// note: 17 stored wires end on pins the file does not list and are not shown
IF NOT (HW_ACV.Mode=Burkert.eACV_Modes.Auto) THEN _w1 := Mix_Status.HW_Valve_Not_Ready; END_IF
Control.Status := _w1;
IF NOT (CW_ACV.Mode=Burkert.eACV_Modes.Auto) THEN _w2 := Mix_Status.CW_Valve_Not_Ready; END_IF
Control.Status := _w2;
Control.Actual_Rate_EU := FIT.Rate;
_w3 := (Control.Mode=Mix_Modes.IDlE) OR (Control.STATUS>Mix_Status.Batch_Ending) OR (Control.Mode=Mix_Modes.Pause);
RATE_PID(
    ACT := FIT.Rate,
    SET := Live_Rate,
    SUP := 0.1,
    OFS := 0.0,
    M_I := 0.0,
    MAN := _w3,
    RST := _w3,
    KP := Control.Config.Flow_KP,
    TN := Control.Config.Flow_TN,
    TV := Control.Config.Flow_TV,
    LL := 0,
    LH := 100.0); // BURKERT_OSCAT_BASIC.CTRL_PID
Control.Flow_CV := RATE_PID.Y;
R_TRIG_2(CLK := _w3 AND (Temperature.Mode.eMode<>Burkert.AIT_Modes.Forced)); // R_Trig
IF R_TRIG_2.Q THEN _w4 := Burkert.AIT_Modes.Alarms_Disabled; END_IF
Temperature.Mode.eMode := _w4;
Control.Actual_Temp_EU := Temperature.EU;
_w5 := (Control.Mode=Mix_Modes.IDlE) OR (Control.Mode=Mix_Modes.Rate_Only) OR (Control.STATUS>Mix_Status.Batch_Ending) OR (Control.STATUS=Mix_Status.Start_Flow) OR (Control.STATUS=Mix_Status.Fit_Reset) OR (Control.Mode=Mix_Modes.Pause);
PID_0(
    ACTUAL := Temperature.EU,
    SET_POINT := Control.Config.TARGET_C,
    KP := Control.Config.Temp_KP,
    TN := Control.Config.Temp_TN,
    TV := Control.Config.Temp_TV,
    Y_MANUAL := 0,
    Y_OFFSET := 0,
    Y_MIN := -100,
    Y_MAX := 100,
    MANUAL := _w5,
    RESET := _w5); // Util.PID
Control.Temp_CV := SEl(Control.Mode=Mix_Modes.Cold_Only, SEl(Control.Mode=Mix_Modes.Hot_Only, PID_0.Y, 100), -100);
SRAMP_0(
    X := Ramp_Target,
    A_UP := Control.Config.Ramp_Rate,
    A_DN := 0-Control.config.Ramp_Rate,
    VU_MAX := Control.config.Max_Flow,
    VD_MAX := 0-Control.config.Max_Flow,
    LIMIT_HIGH := Control.config.Max_Flow,
    LIMIT_LOW := Control.Config.Min_Flow,
    RST := Control.Mode=Mix_Modes.IDlE); // BURKERT_OSCAT_BASIC.SRAMP
Live_Rate := SRAMP_0.Y;
IF Control.Mode=Mix_Modes.IDlE THEN _w6 := Mix_Status.IDle; END_IF
Control.STATUS := _w6;
R_TRIG_0(CLK := (Control.Mode=Mix_Modes.Auto) OR (Control.Mode=Mix_Modes.Hot_Only) OR (Control.Mode=Mix_Modes.Cold_Only) OR (Control.Mode=Mix_Modes.Quick_Start)); // R_Trig
Control.STATUS := SEL(R_TRIG_0.Q, Control.STATUS, Mix_Status.Fit_Reset);
Control.Actual_Volume_EU := FIT.Total;
_w7 := Control.STATUS = Mix_Status.Fit_Reset;
IF _w7 THEN _w8 := False; END_IF
Ramp_active := _w8;
_w9 := NOT (FIT.Total>0.1) AND _w7;
FIT.PLC_Reset := SEL(_w7 AND (FIT.Total>0.1), SEL(_w9, FIT.PLC_Reset, False), True);
_w10 := _w9;
IF _w10 THEN _w11 := Mix_Status.Start_Flow; END_IF
_w12 := _w10;
IF _w12 THEN _w13 := SEL(Control.Mode=Mix_Modes.Hot_Only, _w11, Mix_Status.Temperature_OK); END_IF
IF _w12 THEN _w14 := SEL(Control.Mode=Mix_Modes.Hot_Only, _w13, Mix_Status.Temperature_OK); END_IF
Control.STATUS := _w14;
_w15 := Control.Temp_CV / 100.0;
_w16 := LIMIT(0, Control.Flow_CV * (1.0 + _w15), 100);
Control.HW_CMD := _w16;
HW_ACV.PLC_CMD := _w16;
_w17 := LIMIT(0, Control.Flow_CV * (1.0 - _w15), 100);
Control.CW_CMD := _w17;
CW_ACV.PLC_CMD := _w17;
_w18 := Control.STATUS = Mix_Status.Start_Flow;
IF _w18 THEN _w19 := Control.Config.Min_Flow; END_IF
Ramp_Target := _w19;
TON_0(IN := _w18 AND (Control.Actual_Rate_EU > (Control.Config.Min_Flow*0.8) OR (Control.Mode=Mix_Modes.Quick_Start)), PT := Stage_Delay); // TON
Control.STATUS := SEL(TON_0.Q, Control.STATUS, Mix_Status.Flow_Detected);
TON_1(IN := Control.STATUS = Mix_Status.Flow_Detected, PT := Stage_Delay); // TON
R_TRIG_3(CLK := (Temperature.Mode.eMode<>Burkert.AIT_Modes.Forced) AND TON_1.Q); // R_Trig
IF R_TRIG_3.Q THEN _w20 := Burkert.TT_Modes.Active; END_IF
Temperature.Mode.eMode := _w20;
Control.STATUS := SEL(TON_1.Q, Control.STATUS, Mix_Status.Start_temperature);
Temperature.Burkert.cAlarm_Config.Hi_Hi_Alarm := Control.Config.TARGET_C+(Control.Config.TEMP_WINDOW*4);
Temperature.Burkert.cAlarm_Config.Hi_Warn := Control.Config.TARGET_C+(Control.Config.TEMP_WINDOW*2);
Temperature.Burkert.cAlarm_Config.Low_warn := Control.Config.TARGET_C-(Control.Config.TEMP_WINDOW*2);
Temperature.Burkert.cAlarm_Config.Low_Low_Alarm := Control.Config.TARGET_C-(Control.Config.TEMP_WINDOW*4);
TON_2(IN := Control.STATUS = Mix_Status.Start_temperature AND (Control.Actual_Temp_EU > (Control.Config.TARGET_C-Control.Config.TEMP_WINDOW) OR (Control.Mode=Mix_Modes.Quick_Start)), PT := Stage_Delay); // TON
Control.STATUS := SEL(TON_2.Q, Control.STATUS, Mix_Status.Temperature_OK);
TON_3(IN := Control.STATUS = Mix_Status.Temperature_OK, PT := Stage_Delay); // TON
Control.STATUS := SEL(TON_3.Q, Control.STATUS, Mix_Status.Foundation_Rate);
_w21 := Control.STATUS = Mix_Status.Foundation_Rate;
Ramp_Active := SEL(_w21, Ramp_Active, True);
_w22 := _w21;
IF _w22 THEN _w23 := Control.Config.Foundation_Rate; END_IF
Ramp_Target := _w23;
Control.STATUS := SEL(_w22 AND (Control.Actual_Rate_EU >= (Control.Config.Foundation_Rate*0.9) OR (Control.Mode=Mix_Modes.Quick_Start)), Control.STATUS, Mix_Status.Foundation_Rate_OK);
TON_4(IN := Control.STATUS = Mix_Status.Foundation_Rate_OK AND (FIT.Total >= Control.Config.Foundation_Volume OR (Control.Mode=Mix_Modes.Quick_Start)), PT := Stage_Delay); // TON
Control.STATUS := SEL(TON_4.Q, Control.STATUS, Mix_Status.Foundation_Amount_Complete);
R_TRIG_5(CLK := Control.Mode=Mix_Modes.Resume); // R_trig
TON_5(IN := Control.STATUS = Mix_Status.Foundation_Amount_Complete, PT := Stage_Delay); // TON
Control.STATUS := SEL(R_TRIG_5.Q OR TON_5.Q, Control.STATUS, Mix_Status.Main_Rate);
_w24 := Control.STATUS = Mix_Status.Main_Rate;
R_TRIG_1(CLK := _w24); // R_trig
IF R_TRIG_1.Q THEN _w25 := Control.Actual_Volume_EU; END_IF
Ramp_Start_Volume := _w25;
_w26 := _w24;
IF _w26 THEN _w27 := Control.Config.TARGET_lpm; END_IF
Ramp_Target := _w27;
_w28 := _w26 AND Control.Actual_Rate_EU >= (Control.Config.TARGET_lpm*0.9);
Control.STATUS := SEL(_w28, Control.STATUS, Mix_Status.Main_Rate_OK);
IF _w28 THEN _w29 := Control.Actual_Volume_EU - Ramp_Start_Volume; END_IF
Ramp_Volume := _w29;
_w30 := Control.STATUS = Mix_Status.Main_Rate_OK;
TON_6(IN := _w30, PT := Stage_Delay); // TON
Control.STATUS := SEL(TON_6.Q, Control.STATUS, Mix_Status.Grain_Dispense);
_w31 := Control.STATUS = Mix_Status.Grain_Dispense;
_w32 := _w31;
IF _w32 THEN _w33 := Control.Config.TARGET_C; END_IF
Control.Config.TARGET_C := _w33;
IF _w32 THEN _w34 := Control.Config.TARGET_lpm; END_IF
Ramp_Target := _w34;
Control.STATUS := SEL(_w31 AND Control.Actual_Volume_EU >= (Control.Config.TARGET_L-Control.Config.Foundation_Volume), Control.STATUS, Mix_Status.Batch_Ending);
IF Control.Actual_Rate_EU>0.5 THEN _w35 := ((Control.Config.TARGET_L-Control.Config.Foundation_Volume) - Control.Actual_Volume_EU) / (Control.Actual_Rate_EU/60); END_IF
Control.Grain_ETA_S := REAL_TO_INT(_w35);
_w36 := Control.STATUS = Mix_Status.Batch_Ending;
IF _w36 THEN _w37 := Control.Config.Foundation_Rate; END_IF
Ramp_Target := _w37;
_w38 := (_w24 OR _w30 OR _w31 OR _w36) AND Control.Actual_Volume_EU >= Control.Config.TARGET_L;
Ramp_Active := SEl(_w38, Ramp_Active, FALSE);
Control.STATUS := SEL(_w38, Control.STATUS, Mix_Status.Batch_Complete);
// 0.1: input not connected

END_FUNCTION_BLOCK

// Tempered_Mix_UDFB
FUNCTION_BLOCK Tempered_Mix_UDFB
VAR_INPUT
	//Loop_ID:INT;
END_VAR
VAR_IN_OUT
	HW_ACV:Burkert.cACV;
	CW_ACV:Burkert.cACV;
	Temperature:Burkert.cSensor;
	FIT:Burkert.cFIT;
	Control:Mix_DUT;
END_VAR
VAR_OUTPUT
END_VAR
VAR
	R_TRIG_0: R_Trig;
	RATE_PID: BURKERT_OSCAT_BASIC.CTRL_PID;
	
	Temp_PID: BURKERT_OSCAT_BASIC.CTRL_PID;
	TON_0: TON;
	Stage_Delay: TIME := T#2s;
	TON_1: TON;
	TON_2: TON;
	SRAMP_0: BURKERT_OSCAT_BASIC.SRAMP;
	TON_3: TON;
	TON_4: TON;
	Ramp_Active: BOOL;
	Ramp_Target: REAL;
	TON_5: TON;
	TON_6: TON;
	R_TRIG_1: R_trig;
	Ramp_Start_Volume: REAL;
	Ramp_Volume: REAL;
	R_TRIG_2: R_Trig;
	R_TRIG_3: R_Trig;
	PID_0: Util.PID;
	R_TRIG_4: R_Trig;
	R_TRIG_5:R_trig;
	
	Live_Rate: REAL;
END_VAR
VAR // added by the converter: edge detectors and wires of the graphical bodies
    _w1, _w2, _w3, _w4, _w5, _w6, _w10, _w12, _w13, _w14, _w15, _w16, _w18, _w19, _w21, _w23, _w25, _w30, _w32 : ANY;
    _w7, _w8, _w9, _w11, _w17, _w20, _w22, _w24, _w26, _w28, _w29, _w31, _w33 : BOOL;
    _w27 : REAL;
END_VAR

// note: 18 stored wires end on pins the file does not list and are not shown
IF NOT (HW_ACV.Mode.eMode=Burkert.eACV_Modes.Auto) THEN _w1 := Mix_Status.HW_Valve_Not_Ready; END_IF
Control.Status := _w1;
IF NOT (CW_ACV.Mode.eMode=Burkert.eACV_Modes.Auto) THEN _w2 := Mix_Status.CW_Valve_Not_Ready; END_IF
Control.Status := _w2;
Control.Actual_Rate_EU := FIT.Rate.EU;
_w3 := (Control.Mode=Mix_Modes.IDlE) OR (Control.STATUS>Mix_Status.Batch_Ending) OR (Control.Mode=Mix_Modes.Pause);
RATE_PID(
    ACT := FIT.Rate.EU,
    SET := Live_Rate,
    SUP := 0.1,
    OFS := 0.0,
    M_I := 0.0,
    MAN := _w3,
    RST := _w3,
    KP := Control.Config.Flow_KP,
    TN := Control.Config.Flow_TN,
    TV := Control.Config.Flow_TV,
    LL := 0,
    LH := 100.0); // BURKERT_OSCAT_BASIC.CTRL_PID
Control.Flow_CV := RATE_PID.Y;
R_TRIG_2(CLK := _w3 AND (Temperature.Mode.eMode<>Burkert.AIT_Modes.Forced)); // R_Trig
IF R_TRIG_2.Q THEN _w4 := Burkert.AIT_Modes.Alarms_Disabled; END_IF
Temperature.Mode.eMode := _w4;
Control.Actual_Temp_EU := Temperature.EU;
_w5 := (Control.Mode=Mix_Modes.IDlE) OR (Control.Mode=Mix_Modes.Rate_Only) OR (Control.STATUS>Mix_Status.Batch_Ending) OR (Control.STATUS=Mix_Status.Start_Flow) OR (Control.STATUS=Mix_Status.Fit_Reset) OR (Control.Mode=Mix_Modes.Pause);
PID_0(
    ACTUAL := Temperature.EU,
    SET_POINT := Control.Config.TARGET_C,
    KP := Control.Config.Temp_KP,
    TN := Control.Config.Temp_TN,
    TV := Control.Config.Temp_TV,
    Y_MANUAL := 0,
    Y_OFFSET := 0,
    Y_MIN := -100,
    Y_MAX := 100,
    MANUAL := _w5,
    RESET := _w5); // Util.PID
Control.Temp_CV := SEl(Control.Mode=Mix_Modes.Cold_Only, SEl(Control.Mode=Mix_Modes.Hot_Only, PID_0.Y, 100), -100);
SRAMP_0(
    X := Ramp_Target,
    A_UP := Control.Config.Ramp_Rate,
    A_DN := 0-Control.config.Ramp_Rate,
    VU_MAX := Control.config.Max_Flow,
    VD_MAX := 0-Control.config.Max_Flow,
    LIMIT_HIGH := Control.config.Max_Flow,
    LIMIT_LOW := Control.Config.Min_Flow,
    RST := Control.Mode=Mix_Modes.IDlE); // BURKERT_OSCAT_BASIC.SRAMP
Live_Rate := SRAMP_0.Y;
IF Control.Mode=Mix_Modes.IDlE THEN _w6 := Mix_Status.IDle; END_IF
Control.STATUS := _w6;
R_TRIG_0(CLK := (Control.Mode=Mix_Modes.Auto) OR (Control.Mode=Mix_Modes.Hot_Only) OR (Control.Mode=Mix_Modes.Cold_Only) OR (Control.Mode=Mix_Modes.Quick_Start)); // R_Trig
Control.STATUS := SEL(R_TRIG_0.Q, Control.STATUS, Mix_Status.Fit_Reset);
Control.Actual_Volume_EU := FIT.Total;
_w7 := Control.STATUS = Mix_Status.Fit_Reset;
_w8 := NOT (FIT.Total>0.1) AND _w7;
FIT.PLC_Reset := SEL(_w7 AND (FIT.Total>0.1), SEL(_w8, FIT.PLC_Reset, False), True);
_w9 := _w8;
IF _w9 THEN _w10 := Mix_Status.Start_Flow; END_IF
_w11 := _w9;
IF _w11 THEN _w12 := SEL(Control.Mode=Mix_Modes.Hot_Only, _w10, Mix_Status.Temperature_OK); END_IF
IF _w11 THEN _w13 := SEL(Control.Mode=Mix_Modes.Hot_Only, _w12, Mix_Status.Temperature_OK); END_IF
Control.STATUS := _w13;
_w14 := Control.Temp_CV / 100.0;
_w15 := LIMIT(0, Control.Flow_CV * (1.0 + _w14), 100);
Control.HW_CMD := _w15;
HW_ACV.PLC_CMD := _w15;
_w16 := LIMIT(0, Control.Flow_CV * (1.0 - _w14), 100);
Control.CW_CMD := _w16;
CW_ACV.PLC_CMD := _w16;
_w17 := Control.STATUS = Mix_Status.Start_Flow;
IF _w17 THEN _w18 := Control.Config.Min_Flow; END_IF
Ramp_Target := _w18;
TON_0(IN := _w17 AND (Control.Actual_Rate_EU > (Control.Config.Min_Flow*0.8) OR (Control.Mode=Mix_Modes.Quick_Start)), PT := Stage_Delay); // TON
Control.STATUS := SEL(TON_0.Q, Control.STATUS, Mix_Status.Flow_Detected);
TON_1(IN := Control.STATUS = Mix_Status.Flow_Detected, PT := Stage_Delay); // TON
R_TRIG_3(CLK := (Temperature.Mode.eMode<>Burkert.AIT_Modes.Forced) AND TON_1.Q); // R_Trig
IF R_TRIG_3.Q THEN _w19 := Burkert.TT_Modes.Active; END_IF
Temperature.Mode.iMode := _w19;
Control.STATUS := SEL(TON_1.Q, Control.STATUS, Mix_Status.Start_temperature);
Temperature.Alarm_Config.Setpoints.Hi_Hi_Alarm := Control.Config.TARGET_C+(Control.Config.TEMP_WINDOW*4);
Temperature.Alarm_Config.Setpoints.Hi_Warn := Control.Config.TARGET_C+(Control.Config.TEMP_WINDOW*2);
Temperature.Alarm_Config.Setpoints.Low_Warn := Control.Config.TARGET_C-(Control.Config.TEMP_WINDOW*2);
Temperature.Alarm_Config.Setpoints.Low_Low_Alarm := Control.Config.TARGET_C-(Control.Config.TEMP_WINDOW*4);
TON_2(IN := Control.STATUS = Mix_Status.Start_temperature AND (Control.Actual_Temp_EU > (Control.Config.TARGET_C-Control.Config.TEMP_WINDOW) OR (Control.Mode=Mix_Modes.Quick_Start)), PT := Stage_Delay); // TON
Control.STATUS := SEL(TON_2.Q, Control.STATUS, Mix_Status.Temperature_OK);
TON_3(IN := Control.STATUS = Mix_Status.Temperature_OK, PT := Stage_Delay); // TON
Control.STATUS := SEL(TON_3.Q, Control.STATUS, Mix_Status.Foundation_Rate);
_w20 := Control.STATUS = Mix_Status.Foundation_Rate;
IF _w20 THEN _w21 := Control.Config.Foundation_Rate; END_IF
Ramp_Target := _w21;
Control.STATUS := SEL(_w20 AND (Control.Actual_Rate_EU >= (Control.Config.Foundation_Rate*0.9) OR (Control.Mode=Mix_Modes.Quick_Start)), Control.STATUS, Mix_Status.Foundation_Rate_OK);
TON_4(IN := Control.STATUS = Mix_Status.Foundation_Rate_OK AND (FIT.Total >= Control.Config.Foundation_Volume OR (Control.Mode=Mix_Modes.Quick_Start)), PT := Stage_Delay); // TON
Control.STATUS := SEL(TON_4.Q, Control.STATUS, Mix_Status.Foundation_Amount_Complete);
R_TRIG_5(CLK := Control.Mode=Mix_Modes.Resume); // R_trig
TON_5(IN := Control.STATUS = Mix_Status.Foundation_Amount_Complete, PT := Stage_Delay); // TON
Control.STATUS := SEL(R_TRIG_5.Q OR TON_5.Q, Control.STATUS, Mix_Status.Main_Rate);
_w22 := Control.STATUS = Mix_Status.Main_Rate;
R_TRIG_1(CLK := _w22); // R_trig
IF R_TRIG_1.Q THEN _w23 := Control.Actual_Volume_EU; END_IF
Ramp_Start_Volume := _w23;
_w24 := _w22;
IF _w24 THEN _w25 := Control.Config.TARGET_lpm; END_IF
Ramp_Target := _w25;
_w26 := _w24 AND Control.Actual_Rate_EU >= (Control.Config.TARGET_lpm*0.9);
Control.STATUS := SEL(_w26, Control.STATUS, Mix_Status.Main_Rate_OK);
IF _w26 THEN _w27 := Control.Actual_Volume_EU - Ramp_Start_Volume; END_IF
Ramp_Volume := _w27;
_w28 := Control.STATUS = Mix_Status.Main_Rate_OK;
TON_6(IN := _w28, PT := Stage_Delay); // TON
Control.STATUS := SEL(TON_6.Q, Control.STATUS, Mix_Status.Grain_Dispense);
_w29 := Control.STATUS = Mix_Status.Grain_Dispense;
IF _w29 THEN _w30 := Control.Config.TARGET_lpm; END_IF
Ramp_Target := _w30;
Control.STATUS := SEL(_w29 AND Control.Actual_Volume_EU >= (Control.Config.TARGET_L-Control.Config.Foundation_Volume), Control.STATUS, Mix_Status.Batch_Ending);
Control.Grain_ETA_S := REAL_TO_INT(((Control.Config.TARGET_L-Control.Config.Foundation_Volume) - Control.Actual_Volume_EU) / (Control.Actual_Rate_EU/60));
_w31 := Control.STATUS = Mix_Status.Batch_Ending;
IF _w31 THEN _w32 := Control.Config.Foundation_Rate; END_IF
Ramp_Target := _w32;
_w33 := (_w22 OR _w28 OR _w29 OR _w31) AND Control.Actual_Volume_EU >= Control.Config.TARGET_L;
Ramp_Active := SEl(_w33, Ramp_Active, FALSE);
Control.STATUS := SEL(_w33, Control.STATUS, Mix_Status.Batch_Complete);
// 0.1: input not connected

END_FUNCTION_BLOCK

// Transfer_ACV_FIT_UDFB
FUNCTION_BLOCK Transfer_ACV_FIT_UDFB
VAR_INPUT
	//Index:INT;
	LOCK_OUT:BOOL:=FALSE;
	
END_VAR
VAR_OUTPUT
END_VAR
VAR
	Paused:BOOL;
	Idle_return:BOOL;
	Transfer_Running:BOOL;
	Complete:BOOL;
	ACV_Not_Ready:BOOL;
	//VFD_Not_Ready:BOOL;
	BCV_Not_Ready:BOOL;
	Time_Complete:BOOL;
	FIT_Reset_Complete:BOOL;
	//Pump_Start:BOOL;
	Lockout_Active:BOOL;
	Error:BOOL;
	//Flow_Mode:BOOL;
	Batch_Complete:BOOL;
	//Enable_pump:BOOL;
	
	PID_CV:REAL;
	
	
	
	
	SR2: SR;
	TON_0: TON;
	CTRL_PID_1: BURKERT_OSCAT_BASIC.CTRL_PID;
	R_TRIG_0: R_trig;
	TON_10: TON;
	SR_10: SR;
	RS_11: RS;
	TON_12: TON;
	F_TRIG_10: F_Trig;
	TP11: TP;
END_VAR

VAR_IN_OUT
	Transfer:FIT_VFD_Transfer_DUT;
	//VFD:VFD_Vacon_DUT;
	ACV:ACV_DUT;
	FIT:FIT_DUT;
	
END_VAR
VAR // added by the converter: edge detectors and wires of the graphical bodies
    _w1, _w2, _w6, _w17, _w19 : ANY;
    _w3, _w4, _w5, _w7, _w8, _w9, _w10, _w11, _w12, _w13, _w14, _w15, _w16, _w18, _w20 : BOOL;
END_VAR

